FUNCTION_BLOCK ABSTRACT FB_Handler IMPLEMENTS I_Handler
VAR_INPUT
END_VAR
VAR_OUTPUT
END_VAR
VAR
	iHandler:			I_Handler;
END_VAR

//	The FB_Handler is an abstract function block that implements the I_Handler interface. 
//	It represents a handler in the Chain of Responsibility pattern,
//	where a request can be passed along a chain of potential handlers until one of them handles the request.
//	Each handler in the chain has the ability to either handle the request or pass it to the next handle

METHOD PUBLIC M_Request
VAR_INPUT
	stEvent:			ST_Event;		// event to be handled. 
END_VAR
// The M_Request method is used to handle the request.

IF iHandler <> 0 THEN
	// the request is passed to the next handler 
	iHandler.M_Request(stEvent);
END_IF
END_METHOD

PROPERTY PUBLIC P_Next : I_Handler
GET
P_Next:= iHandler;
END_GET
SET
iHandler:= P_Next;
END_SET
END_PROPERTY

END_FUNCTION_BLOCK

(* stored: Version 1.1.0.1, ProductVersion 3.1.4024.12
   POU FB_Handler: Id {5b555d9d-9f1a-4168-ace2-3a53af448bf3}, SpecialFunc None
   Method M_Request: Id {0dbdffe3-6983-4b80-bcf0-f4c7d261385e}
   Property P_Next: Id {7ff99411-1a84-4185-85aa-4402ac2d8019}
   Get Get: Id {262dea57-9b75-424c-8b01-075b56fa6082}
   Set Set: Id {8eeb1271-99e0-4fef-96c2-4dae70885f83} *)
